TYPE ST_HMI_DataSourceConfig : 
STRUCT
	nID: DINT;
	sDisplayName: WSTRING(80);
	eConfigType: E_SourceType;
	aInputSources: ARRAY [0..0] OF ST_HMI_InputSource;
END_STRUCT
END_TYPE

(* stored: DUT ST_HMI_DataSourceConfig: Id bcafa7ac-0fa5-4e3a-820e-fa2d97b95911 *)
